TYPE SharedContextComSubscribe :
STRUCT
  Region1 : ZApplication.RegionComSubscribe;
  Region2 : ZApplication.RegionComSubscribe;
  Region3 : ZApplication.RegionComSubscribe;
END_STRUCT
END_TYPE

(* stored: Version 1.1.0.1
   DUT SharedContextComSubscribe: Id {f0bb825e-8446-4e84-a3a0-4f05acc1e4f0} *)
